{attribute 'qualified_only'}
VAR_GLOBAL CONSTANT
	pXtsProcessingUnit 			: OTCID	:= 16#01010020;	 
	TRACK_LENGTH 				: LREAL := 7000; // This should be set to the exact length [mm] of the track system
	NUM_MOVERS   				: USINT := 20;   // This should be set to the exact number of movers on the system
	
	// The following should be set to a value **equal to or greater than** the number of objectives needed
	NUM_POSITIONTRIGGERS		: USINT := 10;	// Position Triggers
	NUM_STATIONS				: USINT := 8;	// Stations
	NUM_ZONES					: USINT := 10;	// Zones

	// Station constants
	startStation				: USINT	:= 1;		// set this number to the index of the station all movers should start from
	stationTolerance			: LREAL	:= 1;		// set to number of millimeters tolerance for mover at station
	zeroSpeed					: LREAL	:= 10.0;	// tolerance for definition of not moving
END_VAR

VAR_GLOBAL
	Mover					: ARRAY[1..GVL.NUM_MOVERS] OF Mover;
	Station					: ARRAY[1..GVL.NUM_STATIONS] OF station;
	dsMoverControlFlags		: MoverControlFlags;
END_VAR

(* stored: Version 1.1.0.1, ProductVersion 3.1.4026.8
   GVL GVL: Id {73e6a867-4426-4dae-a583-2a717b275c1c} *)
